// TIA Portal project "Pokayoke_buffer_V13_SP1_V15" (V15)
// Software para controle  da altura do empilhamento das caixas no espelho da estufagem do "KD".

(* hardware
DEVICE "S7-1200 station_1"  S7-1200 Station
   slot 0: "Rack_0"  Rack  V1.0
   slot 1: "PLC_Automation"  CPU 1214C DC/DC/DC  6ES7 214-1AG40-0XB0  V4.0
*)

// ===== PLC "PLC_Automation"  CPU 1214C DC/DC/DC =====

VAR_GLOBAL   // PLC tag table "Default tag table"
   "Clock_10Hz" AT %M0.0 : Bool;   // Pulsos automáticos de (0.1 segundo)
   "Clock_5Hz" AT %M0.1 : Bool;   // Pulsos automáticos de (0.2 segundo)
   "Clock_2.5Hz" AT %M0.2 : Bool;   // Pulsos automáticos de (0.4 segundo)
   "Clock_2Hz" AT %M0.3 : Bool;   // Pulsos automáticos de (0.5 segundo)
   "Clock_1.25Hz" AT %M0.4 : Bool;   // Pulsos automáticos de (0.8 segundo)
   "Clock_1Hz" AT %M0.5 : Bool;   // Pulsos automáticos de (1 segundo)
   "Clock_0.625Hz" AT %M0.6 : Bool;   // Pulsos automáticos de (1.6 segundos)
   "Clock_0.5Hz" AT %M0.7 : Bool;   // Pulsos automáticos de (2 segundos)
END_VAR

VAR_GLOBAL   // PLC tag table "Peripheral_inputs"
   "P.IN_Signal_Scanner" AT %I0.0 : Bool;   // Sinal de Leitura de obstáculo do Scanner.
END_VAR

VAR_GLOBAL   // PLC tag table "Peripheral_outputs"
   "P.OUT_Buzzer" AT %Q0.0 : Bool;   // Sinal para ligar a Sirene de aviso de obstáculo no scanner.
   "P.OUT_GreenLight" AT %Q0.1 : Bool;   // Sinal para ligar a Lâmpada verde.
   "P.OUT_RedLight" AT %Q0.2 : Bool;   // Sinal para ligar a Lâmpada vermelha.
END_VAR

// folder: DBs/FBs

DATA_BLOCK "Scanner_espelho_DB_FB1"   // DB10
{ S7_Optimized_Access := 'FALSE' }
VERSION : 0.1
// stored: InstanceOfName Scanner_espelho
"Scanner_espelho"
BEGIN
END_DATA_BLOCK

// folder: DBs_IHM

DATA_BLOCK "IHM_Signals"   // DB5
{ S7_Optimized_Access := 'FALSE' }
VERSION : 0.1
   VAR
      "M.S_Enable.Scanner" : Bool;   // Sinal da IHM para liberar o funcionamento da lógica de monitoramento do Scanner.
      Empty1 : Bool;
      Empty2 : Bool;
      Empty3 : Bool;
      Empty4 : Bool;
      Empty5 : Bool;
      Empty6 : Bool;
      Empty7 : Bool;
   END_VAR
BEGIN
END_DATA_BLOCK

// folder: DBs_System

DATA_BLOCK "System_IN"   // DB3
{ S7_Optimized_Access := 'FALSE' }
VERSION : 0.1
BEGIN
END_DATA_BLOCK

DATA_BLOCK "System_OUT"   // DB4
{ S7_Optimized_Access := 'FALSE' }
VERSION : 0.1
   VAR
      "M.S_YellowScreen" : Bool;   // Memória com o sinal para a Tela da linha "ECU" ficar amarela.
      "M.S_RedScreen" : Bool;   // Memória com o sinal para a Tela da linha "ECU" ficar Vermelha.
      Empty : Bool;
      "M.S_StopLine" : Bool;   // Memória com o sinal para bloqueio da linha de "ECU".
      Emtpy1 : Bool;
      Emtpy2 : Bool;
      Emtpy3 : Bool;
      Empty4 : Bool;
   END_VAR
BEGIN
END_DATA_BLOCK

// folder: DBs_peripheral_signals

DATA_BLOCK "Peripheral_signals.IN"   // DB1
{ S7_Optimized_Access := 'TRUE' }
VERSION : 0.1
   VAR
      "M.S_Signal_Scanner" : Bool;   // Memória de movimentação do sinal de obstáculo no Scanner.
   END_VAR
BEGIN
END_DATA_BLOCK

DATA_BLOCK "Peripheral_signals.OUT"   // DB2
{ S7_Optimized_Access := 'TRUE' }
VERSION : 0.1
   VAR
      "M.S_Buzzer" : Bool;   // Memória de movimentação do sinal de "Liga Sirene".
      "M.S_GreenLight" : Bool;   // Memória de movimentação do sinal de "Liga lâmpada verde".
      "M.S_RedLight" : Bool;   // Memória de movimentação do sinal de "Liga lâmpada vermelha".
   END_VAR
BEGIN
END_DATA_BLOCK

// folder: (top level)

ORGANIZATION_BLOCK "Main"   // OB1, LAD, ProgramCycle
TITLE = "Main Program Sweep (Cycle)"
{ S7_Optimized_Access := 'TRUE' }
VERSION : 0.1
   VAR_INPUT
      Initial_Call : Bool;   // Initial call of this OB
      Remanence : Bool;   // =True, if remanent data are available
   END_VAR
BEGIN

REGION Network 1: Peripheral input signals.
   // Tranferência dos sinais periféricos de entrada para as memórias de movimentação dos sinais de entrada.
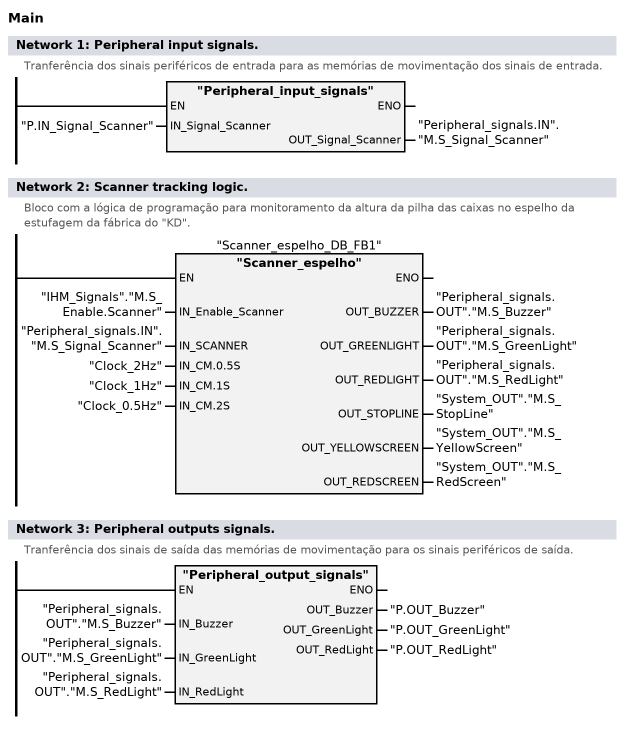
   RUNG wire#powerrail
      "Peripheral_input_signals"(IN_Signal_Scanner := "P.IN_Signal_Scanner", OUT_Signal_Scanner => "Peripheral_signals.IN"."M.S_Signal_Scanner")
   END_RUNG
   // the same network as SCL:
   "Peripheral_input_signals"(IN_Signal_Scanner := "P.IN_Signal_Scanner",
                           OUT_Signal_Scanner => "Peripheral_signals.IN"."M.S_Signal_Scanner");
END_REGION

REGION Network 2: Scanner tracking logic.
   // Bloco com a lógica de programação para monitoramento da altura da pilha das caixas no espelho da estufagem da fábrica do "KD".
   RUNG wire#powerrail
      "Scanner_espelho_DB_FB1"(IN_Enable_Scanner := "IHM_Signals"."M.S_Enable.Scanner", IN_SCANNER := "Peripheral_signals.IN"."M.S_Signal_Scanner", "IN_CM.0.5S" := "Clock_2Hz", "IN_CM.1S" := "Clock_1Hz", "IN_CM.2S" := "Clock_0.5Hz", OUT_BUZZER => "Peripheral_signals.OUT"."M.S_Buzzer", OUT_GREENLIGHT => "Peripheral_signals.OUT"."M.S_GreenLight", OUT_REDLIGHT => "Peripheral_signals.OUT"."M.S_RedLight", OUT_STOPLINE => "System_OUT"."M.S_StopLine", OUT_YELLOWSCREEN => "System_OUT"."M.S_YellowScreen", OUT_REDSCREEN => "System_OUT"."M.S_RedScreen")
   END_RUNG
   // the same network as SCL:
   "Scanner_espelho_DB_FB1"(IN_Enable_Scanner := "IHM_Signals"."M.S_Enable.Scanner",   // "Scanner_espelho"
                           IN_SCANNER := "Peripheral_signals.IN"."M.S_Signal_Scanner",
                           "IN_CM.0.5S" := "Clock_2Hz",
                           "IN_CM.1S" := "Clock_1Hz",
                           "IN_CM.2S" := "Clock_0.5Hz",
                           OUT_BUZZER => "Peripheral_signals.OUT"."M.S_Buzzer",
                           OUT_GREENLIGHT => "Peripheral_signals.OUT"."M.S_GreenLight",
                           OUT_REDLIGHT => "Peripheral_signals.OUT"."M.S_RedLight",
                           OUT_STOPLINE => "System_OUT"."M.S_StopLine",
                           OUT_YELLOWSCREEN => "System_OUT"."M.S_YellowScreen",
                           OUT_REDSCREEN => "System_OUT"."M.S_RedScreen");
END_REGION

REGION Network 3: Peripheral outputs signals.
   // Tranferência dos sinais de saída das memórias de movimentação para os sinais periféricos de saída.
   RUNG wire#powerrail
      "Peripheral_output_signals"(IN_Buzzer := "Peripheral_signals.OUT"."M.S_Buzzer", IN_GreenLight := "Peripheral_signals.OUT"."M.S_GreenLight", IN_RedLight := "Peripheral_signals.OUT"."M.S_RedLight", OUT_Buzzer => "P.OUT_Buzzer", OUT_GreenLight => "P.OUT_GreenLight", OUT_RedLight => "P.OUT_RedLight")
   END_RUNG
   // the same network as SCL:
   "Peripheral_output_signals"(IN_Buzzer := "Peripheral_signals.OUT"."M.S_Buzzer",
                           IN_GreenLight := "Peripheral_signals.OUT"."M.S_GreenLight",
                           IN_RedLight := "Peripheral_signals.OUT"."M.S_RedLight",
                           OUT_Buzzer => "P.OUT_Buzzer",
                           OUT_GreenLight => "P.OUT_GreenLight",
                           OUT_RedLight => "P.OUT_RedLight");
END_REGION
END_ORGANIZATION_BLOCK

// folder: FBs

FUNCTION_BLOCK "Scanner_espelho"   // FB1, SCL
{ S7_Optimized_Access := 'FALSE' }
VERSION : 0.1
   VAR_INPUT
      IN_Enable_Scanner : Bool;   // Habilita Scanner pela IHM.
      IN_SCANNER : Bool;   // Sinal de monitoramento do Scanner.
      "IN_CM.0.5S" : Bool;   // Sinal "Clock memory" de 0,5 segundos para a sirene.
      "IN_CM.1S" : Bool;   // Sinal "Clock memory" de 1 segundo para a sirene.
      "IN_CM.2S" : Bool;   // Sinal "Clock memory" de 2 segundos para o Led vermelho.
   END_VAR
   VAR_OUTPUT
      OUT_BUZZER : Bool;   // Sirene para alerta sonoro.
      OUT_GREENLIGHT : Bool;   // Lâmpada verde para alerta de situação no padrão.
      OUT_REDLIGHT : Bool;   // Lâmpada vermelha para alerta de situação fora do padrão.
      OUT_STOPLINE : Bool;   // Sinal para bloqueio da linha de ECU.
      OUT_YELLOWSCREEN : Bool;   // Sinal para a TV da linha ECU Ficar com a Tela amarela.
      OUT_REDSCREEN : Bool;   // Sinal para a TV da linha ECU Ficar com a Tela vermelha.
   END_VAR
   VAR
      S_TIMER_SCANNER : TON_TIME;   // Timer conta 25s
      "S_TIMER_SCANNER.IN" : Bool;   // Memória liga o timer.
      S_SEQUENCE : Int;   // memória para atribuir as sequências.
      "S_GREEN.LIGHT_1" : Bool;   // Auxiliar lâmpada verde.
      "S_RED.LIGHT_1" : Bool;   // Auxiliar lâmpada vermelha.
      S_BUZZER_1 : Bool;   // Auxiliar Sirene.
      S_YELLOWSCREEN : Bool;   // Auxiliar tela amarela.
      S_REDSCREEN : Bool;   // Auxiliar tela vermelha.
      S_STOPLINE : Bool;   // Auxiliar para a linha de ECU.
   END_VAR
BEGIN
   // GOD BE PRAISED

   //READ INFORMATION
   #"S_TIMER_SCANNER.IN" := #IN_SCANNER AND #IN_Enable_Scanner;

   //TIMER
   #S_TIMER_SCANNER(IN := #"S_TIMER_SCANNER.IN",
                    PT := T#25S);

   //1º CONDITION (ENABLE_SCANNER := OFF)
   IF NOT #IN_Enable_Scanner THEN
     #S_SEQUENCE := 1;
   END_IF;

   //2º CONDITION (SCANNER := OFF)
   IF NOT #IN_SCANNER AND #IN_Enable_Scanner THEN
     #S_SEQUENCE := 2;
   END_IF;

   //3º CONDITION (SCANNER := ON FROM 0 TO 10S)
   IF (#S_TIMER_SCANNER.ET > T#0S) AND
     (#S_TIMER_SCANNER.ET <= T#10S) THEN
     #S_SEQUENCE := 3;
   END_IF;

   //4º CONDITION (SCANNER := ON FROM 11 TO 24S)
   IF (#S_TIMER_SCANNER.ET > T#10S) AND
     (#S_TIMER_SCANNER.ET < T#25S) THEN
     #S_SEQUENCE := 4;
   END_IF;

   //5º CONDITION (SCANNER := ON MORE THAN 25S)
   IF #S_TIMER_SCANNER.Q THEN
     #S_SEQUENCE := 5;
   END_IF;

   CASE #S_SEQUENCE OF
     1:  // GREEN LIGHT := ON AND CM 1S || RED LIGHT := ON AND CM 1S || BUZZER := OFF || YELLOWSCREEN := OFF || REDSCREEN := OFF
       #"S_GREEN.LIGHT_1" := #"IN_CM.1S";
       #"S_RED.LIGHT_1" := #"IN_CM.1S";
       #S_BUZZER_1 := 0;
       #S_YELLOWSCREEN := 0;
       #S_REDSCREEN := 0;
       #S_STOPLINE := 0;

     2:  // GREEN LIGHT := ON || RED LIGHT := OFF || BUZZER := OFF || YELLOWSCREEN := OFF || REDSCREEN := OFF
       #"S_GREEN.LIGHT_1" := 1;
       #"S_RED.LIGHT_1" := 0;
       #S_BUZZER_1 := 0;
       #S_YELLOWSCREEN := 0;
       #S_REDSCREEN := 0;
       #S_STOPLINE := 0;

     3:  // GREEN LIGHT := ON || RED LIGHT := ON || BUZZER := OFF
       #"S_GREEN.LIGHT_1" := 0;
       #"S_RED.LIGHT_1" := 1;
       #S_BUZZER_1 := 0;
       #S_YELLOWSCREEN := 0;
       #S_REDSCREEN := 0;
       #S_STOPLINE := 0;

     4:  // GREEN LIGHT := OFF || RED LIGHT := ON AND CM 1S || BUZZER := ON AND CM 1S || YELLOWSCREEN := ON
       #"S_GREEN.LIGHT_1" := 0;
       #"S_RED.LIGHT_1" := #"IN_CM.2S";
       #S_BUZZER_1 := #"IN_CM.1S";
       #S_YELLOWSCREEN := 1;
       #S_REDSCREEN := 0;
       #S_STOPLINE := 0;

     5:  // GREEN LIGHT := OFF || RED LIGHT := ON || BUZZER := ON AND CM 0.5S || STOPLINE := ON || REDSCREEN := ON || YELLOWSCREEN := OFF
       #"S_GREEN.LIGHT_1" := 0;
       #"S_RED.LIGHT_1" := 1;
       #S_BUZZER_1 := #"IN_CM.0.5S";
       #S_YELLOWSCREEN := 0;
       #S_REDSCREEN := 1;
       #S_STOPLINE := 1;

   END_CASE;


   //SET OUT INFORMATION
   #OUT_BUZZER := #S_BUZZER_1;
   #OUT_GREENLIGHT := #"S_GREEN.LIGHT_1";
   #OUT_REDLIGHT := #"S_RED.LIGHT_1";
   #OUT_REDSCREEN := #S_REDSCREEN;
   #OUT_STOPLINE := #S_STOPLINE;
   #OUT_YELLOWSCREEN := #S_YELLOWSCREEN;
END_FUNCTION_BLOCK

// folder: FCs

FUNCTION "Peripheral_input_signals" : Void   // FC1, SCL
{ S7_Optimized_Access := 'TRUE' }
VERSION : 0.1
   VAR_INPUT
      IN_Signal_Scanner : Bool;   // Sinal de obstáculo do Scanner.
   END_VAR
   VAR_OUTPUT
      OUT_Signal_Scanner : Bool;   // Sinal de obstáculo do Scanner para a memória de movimentação.
   END_VAR
BEGIN
   // Peripheral Input/ Memory Input

   #OUT_Signal_Scanner := #IN_Signal_Scanner;
   //___________________________________________________________________________________________________________________________________________________________________________________________________________________
END_FUNCTION

FUNCTION "Peripheral_output_signals" : Void   // FC2, SCL
{ S7_Optimized_Access := 'TRUE' }
VERSION : 0.1
   VAR_INPUT
      IN_Buzzer : Bool;   // Sinal da memória de movimentação "Liga Sirene".
      IN_GreenLight : Bool;   // Sinal da memória de movimentação "Liga lâmpada verde".
      IN_RedLight : Bool;   // Sinal da memória de movimentação "Liga lâmpada vermelha".
   END_VAR
   VAR_OUTPUT
      OUT_Buzzer : Bool;   // Sinal para saída periférica de "Liga Sirene".
      OUT_GreenLight : Bool;   // Sinal para saída periférica de "Liga lâmpada verde".
      OUT_RedLight : Bool;   // Sinal para saída periférica de "Liga lâmpada vermelha".
   END_VAR
BEGIN
   // Memory Output/Peripheral Output

   #OUT_Buzzer := #IN_Buzzer;
   #OUT_GreenLight := #IN_GreenLight;
   #OUT_RedLight := #IN_RedLight;
   //___________________________________________________________________________________________________________________________________________________________________________________________________________________
END_FUNCTION